Fanuc KAREL source: kt00410.KL

-- PROVISIONAL review KL for V770-1; original PC SHA256 4b1b6fd8c59d87b3b7a045031e596dd530a3c68b140e660ccee243a9bdc1c519
-- Incomplete behavior may be omitted. Consult companion uncertainty JSON. Do not deploy.
PROGRAM KT00410
%NOLOCKGROUP
VAR
  S1 : STRING[80]
  S2 : STRING[80]
  OUT : BOOLEAN
BEGIN
  -- UNRESOLVED_PC offsets 5-14; opcodes 3F,75
  -- UNRESOLVED_PC offsets 19-28; opcodes 3F,75
  -- UNRESOLVED_PC offsets 33-42; opcodes 3F,75
  -- UNRESOLVED_PC offsets 47-56; opcodes 3F,75
  -- UNRESOLVED_PC offsets 61-80; opcodes 73,73,87,23
  -- UNRESOLVED_PC offsets 85-89; opcodes 7F
END KT00410
